// TwinCAT 3 PLC project CommonLibrary
// ProgramVersion: 3.1.4023.0
// libraries:
//   Tc2_Standard, * (Beckhoff Automation GmbH)
//   Tc2_System, * (Beckhoff Automation GmbH)
// project tree:
//   / GVL_Param.TcGVL
//   HMI/Button/DUTs/ E_Hmi_ButtonBehaviour.TcDUT, S_Hmi_Button.TcDUT
//   HMI/Button/ FB_Hmi_Button.TcPOU
//   HMI/Led/DUTs/ E_Hmi_LedColor.TcDUT, S_Hmi_Led.TcDUT
//   HMI/Led/ FB_Hmi_Led.TcPOU
//   HMI/Switch/ FB_Hmi_Switch.TcPOU (not stored)
//   Utilities/DUTs/ LoopIterator.TcDUT (not stored)
//   Utilities/InitializeControl/ ASSERT.TcPOU, FB_InitializeControl.TcPOU (not stored)
//   Utilities/Timers/ FB_Timer.TcPOU, FB_TimerManager.TcPOU, I_Timer.TcIO, TIMERS.TcGVL (not stored)

// ---- HMI/Button/DUTs/E_Hmi_ButtonBehaviour.TcDUT
{attribute 'qualified_only'}
{attribute 'strict'}
TYPE E_Hmi_ButtonBehaviour :
(
	MomentaryOn := 0,
	MomentaryOff := 1,
	Toggle := 2,
	Set := 3,
	Reset := 4
)UINT;
END_TYPE

// ---- HMI/Button/DUTs/S_Hmi_Button.TcDUT
TYPE S_Hmi_Button :
STRUCT
	Click: BOOL;
	Enabled: BOOL;
	Visibility: BOOL;
	Led: S_Hmi_Led;
END_STRUCT
END_TYPE

// ---- HMI/Led/DUTs/E_Hmi_LedColor.TcDUT
{attribute 'qualified_only'}
{attribute 'strict'}
TYPE E_Hmi_LedColor :
(
	Yellow := 0,
	YellowGreen := 1,
	Green := 2,
	BlueGreen := 3,
	Blue := 4,
	BlueViolet := 5,
	Violet := 6,
	RedViolet := 7,
	Red := 8,
	RedOrange := 9,
	Orange := 10,
	YellowOrange := 11,
	White := 12,
	Gray := 13,
	Black := 14,
	Blank := 15
)UINT;
END_TYPE

// ---- HMI/Led/DUTs/S_Hmi_Led.TcDUT
TYPE S_Hmi_Led :
STRUCT
	OnOff: BOOL;
	OnColor: UINT;
	OffColor: UINT;
	Visibility: BOOL;
END_STRUCT
END_TYPE

// ---- GVL_Param.TcGVL
VAR_GLOBAL CONSTANT
	MAX_INIT_LIST: INT := 64;
END_VAR

// ---- Utilities/Timers/I_Timer.TcIO
INTERFACE I_Timer

METHOD Execute
END_METHOD

METHOD Register
END_METHOD

END_INTERFACE

// ---- HMI/Button/FB_Hmi_Button.TcPOU
FUNCTION_BLOCK FB_Hmi_Button
VAR
	_rButton: REFERENCE TO S_Hmi_Button;

	_Led: FB_Hmi_Led;

	_behaviour: E_Hmi_ButtonBehaviour;
	_value: BOOL;

	_initialized: BOOL;
END_VAR

IF _initialized THEN
	IF _behaviour = E_Hmi_ButtonBehaviour.MomentaryOff THEN
		_value := TRUE;
	ELSIF _behaviour = E_Hmi_ButtonBehaviour.MomentaryOn THEN
		_value := FALSE;
	END_IF

	IF _rButton.Click THEN
		CASE _behaviour OF
			E_Hmi_ButtonBehaviour.MomentaryOff:
				Reset();

			E_Hmi_ButtonBehaviour.MomentaryOn:
				Set();

			E_Hmi_ButtonBehaviour.Reset:
				Reset();

			E_Hmi_ButtonBehaviour.Set:
				Set();

			E_Hmi_ButtonBehaviour.Toggle:
				Toggle();
		END_CASE

		_rButton.Click := FALSE;
	END_IF
END_IF

PROPERTY PUBLIC Enabled : BOOL
SET
_rButton.Enabled := Enabled;
END_SET
END_PROPERTY

METHOD PUBLIC Initialize : BOOL
VAR_INPUT
	rButton: REFERENCE TO S_Hmi_Button;
	behaviour: E_Hmi_ButtonBehaviour;
END_VAR
IF __ISVALIDREF(rButton) THEN
	_Led.initialize(rButton.Led);
	_rButton REF= rButton;
	_behaviour := behaviour;

	_initialized := Initialize := TRUE;
END_IF
END_METHOD

PROPERTY PUBLIC Led : POINTER TO FB_Hmi_Led;
GET
Led := ADR(_Led);
END_GET
END_PROPERTY

METHOD PUBLIC Reset
IF _initialized AND_THEN _rButton.Enabled THEN
	_value := FALSE;
END_IF
END_METHOD

METHOD PUBLIC Set
IF _initialized AND_THEN _rButton.Enabled THEN
	_value := TRUE;
END_IF
END_METHOD

METHOD PUBLIC Toggle
IF _initialized AND_THEN _rButton.Enabled THEN
	_value := NOT _value;
END_IF
END_METHOD

PROPERTY PUBLIC Value : BOOL
GET
Value := _value;
END_GET
END_PROPERTY

PROPERTY PUBLIC Visibility : BOOL
SET
IF _initialized THEN
	_rButton.Visibility := Visibility;
END_IF
END_SET
END_PROPERTY

END_FUNCTION_BLOCK

// ---- HMI/Led/FB_Hmi_Led.TcPOU
FUNCTION_BLOCK FB_Hmi_Led
VAR
	_rLed: REFERENCE TO S_Hmi_Led;

	_blink: BOOL;
	_blinkTime: TIME;
	_Blinker: FB_Timer;

	_initialized: BOOL;
END_VAR

IF _blink THEN
	IF _Blinker.Done THEN
		_Blinker.Start(_blinkTime);
		_rLed.OnOff := NOT _rLed.OnOff;
	END_IF

	_Blinker();
END_IF

PROPERTY PUBLIC Blink : BOOL
SET
_blink := Blink;
_rLed.OnOff := FALSE;
END_SET
END_PROPERTY

PROPERTY PUBLIC BlinkTime : TIME
SET
BlinkTime := _blinkTime;
END_SET
END_PROPERTY

METHOD PUBLIC Initialize : BOOL
VAR_INPUT
	rLed: REFERENCE TO S_Hmi_Led;
END_VAR
IF __ISVALIDREF(rLed) THEN
	_rLed REF= rLed;
	_initialized := Initialize := TRUE;
END_IF
END_METHOD

PROPERTY PUBLIC OffColor : UINT
SET
_rLed.OffColor := OffColor;
END_SET
END_PROPERTY

PROPERTY PUBLIC OnColor : UINT
SET
_rLed.OnColor := OnColor;
END_SET
END_PROPERTY

PROPERTY PUBLIC OnOff : BOOL
SET
_rLed.OnOff := OnOff;
END_SET
END_PROPERTY

PROPERTY PUBLIC Visibility : BOOL
SET
_rLed.Visibility := Visibility;
END_SET
END_PROPERTY

END_FUNCTION_BLOCK

// ---- Utilities/Timers/FB_Timer.TcPOU
FUNCTION_BLOCK FB_Timer IMPLEMENTS I_Timer
VAR
	_Timer: TON;

	_done: BOOL;
	_busy: BOOL;
	_free: BOOL := TRUE;
END_VAR

PROPERTY PUBLIC Busy : BOOL
GET
Busy := _busy;
END_GET
END_PROPERTY

PROPERTY PUBLIC Done : BOOL
GET
Done := _done;
END_GET
END_PROPERTY

PROPERTY PUBLIC ElapsedTime : TIME
GET
ElapsedTime := _Timer.ET;
END_GET
END_PROPERTY

METHOD Execute
_Timer();

IF _Timer.Q THEN
	_done := TRUE;
	_busy := FALSE;
END_IF
END_METHOD

METHOD Register : BOOL
VAR_INPUT
	Timer: I_Timer;
END_VAR
Register := TIMERS.Manager.Register(THIS^);
END_METHOD

METHOD PUBLIC Reset
_Timer(IN := FALSE);

_done := FALSE;
_busy := FALSE;
_free := TRUE;
END_METHOD

METHOD PUBLIC Start
VAR_INPUT
	delay: TIME;
END_VAR
IF _free THEN
	_Timer(IN := FALSE);
	_Timer(IN := TRUE,
			PT := delay);

	_busy := TRUE;
	_done := FALSE;
	_free := FALSE;
END_IF
END_METHOD

END_FUNCTION_BLOCK

// ---- Utilities/InitializeControl/ASSERT.TcPOU
FUNCTION ASSERT : BOOL
VAR_INPUT
	passed: BOOL;
	text: STRING;
END_VAR
VAR
END_VAR

IF NOT passed THEN
	ADSLOGSTR(msgCtrlMask := ADSLOG_MSGTYPE_ERROR, msgFmtStr := 'FAILED: %s', text);
END_IF

// Return the result of the assertion for further processing
ASSERT := passed;

END_FUNCTION

// ---- Utilities/Timers/FB_TimerManager.TcPOU
FUNCTION_BLOCK FB_TimerManager
VAR
	_aTimers: ARRAY [1..TIMERS.MAX_TIMER] OF I_Timer;
	_count: INT;
END_VAR

FOR

METHOD PUBLIC Register : BOOL
VAR_INPUT
	Timer: I_Timer;
END_VAR
END_METHOD

END_FUNCTION_BLOCK
